FUNCTION_BLOCK FB_MoveSingleaxis_Case
VAR_INPUT
	///run cyclic
	bStart: BOOL;
END_VAR
VAR_OUTPUT
	bBusy: BOOL;
	bErr: BOOL;
	nErrorID: UDINT;
END_VAR
VAR
	Pos_a: REAL := 100;
	Velo_a: REAL := 50;

	Pos_b: REAL := 200;
	Velo_b: REAL := 40;

	///FB Instances
	AxMc_MoveAbsolut1: MC_MoveAbsolute;
	AxMcMoveAbsolut1Out: ST_McOutputs;
	
	StartTrig: R_TRIG;
	nstate: INT;
	nLaststate: INT;
END_VAR
VAR_IN_OUT
	stAxisRef: AXIS_REF;
END_VAR


StartTrig(CLK:=bStart , Q=> );
CASE nstate OF

0: 	(*INIT*)
	bBusy :=FALSE;
	IF bStart AND StartTrig.Q THEN
		bErr := FALSE;
		nErrorID :=0;
		bBusy :=TRUE;
		nLastState :=0;
		nstate:=10;
	END_IF
10: 	(*Set Parameters for MC Block for positioning a *)
		AxMc_MoveAbsolut1.Position := Pos_a ;
		AxMc_MoveAbsolut1.Velocity := Velo_a ;
		AxMc_MoveAbsolut1.Execute := TRUE;
		IF AxMc_MoveAbsolut1.Done AND bStart THEN
			AxMc_MoveAbsolut1.Execute := FALSE;
			nstate := 40;
		ELSIF AxMc_MoveAbsolut1.Error OR AxMc_MoveAbsolut1.CommandAborted THEN
			nErrorID := AxMc_MoveAbsolut1.ErrorID;
			bErr := TRUE;
			nLastState := nstate;
			nstate := 1000;
		END_IF


40: 	(*Set Parameters for MC Block for positioning a *)
		AxMc_MoveAbsolut1.Position := Pos_b ;
		AxMc_MoveAbsolut1.Velocity := Velo_b ;
		AxMc_MoveAbsolut1.Execute := TRUE;

		IF AxMc_MoveAbsolut1.Done AND bStart THEN
			AxMc_MoveAbsolut1.Execute := FALSE;
			nstate := 10;
		ELSIF AxMc_MoveAbsolut1.Error OR AxMc_MoveAbsolut1.CommandAborted THEN
			nErrorID := AxMc_MoveAbsolut1.ErrorID;
			bErr := TRUE;
			nLastState := nstate;
			nstate := 1000;
		END_IF


1000: 	(*Errorstate*)
		//nLastState; (*For Debug*)
		//nErrorID;
		AxMc_MoveAbsolut1.Execute := FALSE;
		IF NOT bStart  THEN
			nstate := nLastState;
		END_IF


END_CASE
actFBCalls();

ACTION actFBCalls:
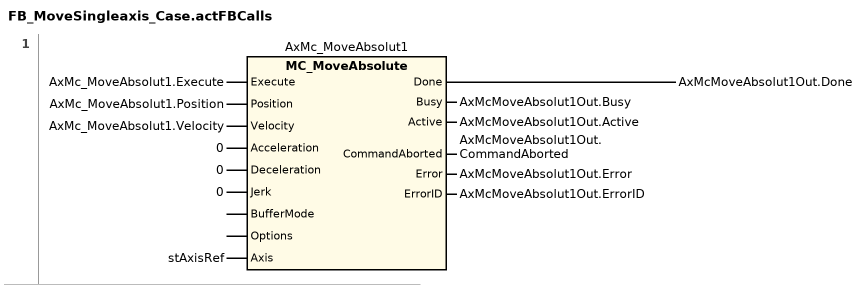
// NETWORK 1
AxMc_MoveAbsolut1(
    Execute := AxMc_MoveAbsolut1.Execute,
    Position := AxMc_MoveAbsolut1.Position,
    Velocity := AxMc_MoveAbsolut1.Velocity,
    Acceleration := 0,
    Deceleration := 0,
    Jerk := 0,
    Axis := stAxisRef,
    Busy => AxMcMoveAbsolut1Out.Busy,
    Active => AxMcMoveAbsolut1Out.Active,
    CommandAborted => AxMcMoveAbsolut1Out.CommandAborted,
    Error => AxMcMoveAbsolut1Out.Error,
    ErrorID => AxMcMoveAbsolut1Out.ErrorID); // MC_MoveAbsolute
AxMcMoveAbsolut1Out.Done := AxMc_MoveAbsolut1.Done;
END_ACTION

END_FUNCTION_BLOCK

(* stored: Version 1.1.0.1, ProductVersion 3.1.4022.17
   POU FB_MoveSingleaxis_Case: Id {de27a99e-cc7d-4c01-bd8f-1d193f3543d2}, SpecialFunc None
   Action actFBCalls: Id {a48fc8eb-5868-43a9-bcda-9bea56bc58b0} *)
